FUNCTION_BLOCK AX_E_PERMIT (* permissive propagation of an event *)
  (* Standard: 61499-1 Annex A; Description: Copyright (c) 2017 fortiss GmbH, HR Agrartechnik GmbH This program and the accompanying materials are made available under the terms of the Eclipse Public License 2.0 which is available at https://www.eclipse.org/legal/epl-2.0/ SPDX-License-Identifier: EPL-2.0 *)
  (* Version 3.0, 2025-04-14, Patrick Aigner, changed package *)
  (* Version 1.0, 2017-09-20, Alois Zoitl, fortiss GmbH, initial API and implementation and/or initial documentation *)
  PACKAGE adapter::events::unidirectional;
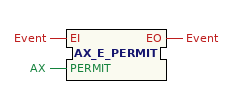
  EVENT_INPUT
    EI; (* Event input *)
  END_EVENT
  EVENT_OUTPUT
    EO; (* Event output *)
  END_EVENT
  SOCKETS
    PERMIT : adapter::types::unidirectional::AX; (* Event input *)
  END_SOCKETS
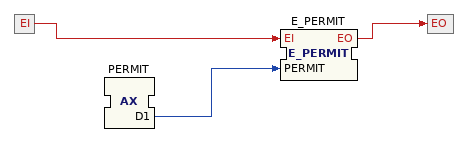
  FBS
    E_PERMIT : iec61499::events::E_PERMIT;
  END_FBS
  EVENT_CONNECTIONS
    E_PERMIT.EO TO EO;
    EI TO E_PERMIT.EI;
  END_CONNECTIONS
  DATA_CONNECTIONS
    PERMIT.D1 TO E_PERMIT.PERMIT;
  END_CONNECTIONS
END_FUNCTION_BLOCK
